{attribute 'GeneratedUsingTerminal: EL3024-0000-0019'}
{attribute addProperty BoxType "EL3024-0000-0019"}
{attribute addProperty Id "ValueAT %I*INT2"}
{attribute addProperty CRC "2162654570"}
{attribute addProperty Size "2"}
TYPE AI_Compact_Channel_80E77D6A :
STRUCT
	{attribute addProperty Name "Value"}
	Value AT %I* : INT;
END_STRUCT
END_TYPE

(* stored: Version 1.2.0.0, ProductVersion 3.1.4024.9
   DUT AI_Compact_Channel_80E77D6A: Id {16efbe88-5bc7-4fc4-8dc4-fc88f61d9097} *)
